Staubli VAL3: loadPage.pgx

program loadPage(string x_sPage, string& x_sItems[])
// load the next page
  local num i
begin
  // look if the page libload is correct
  i=page:libLoad(x_sPage)
  delay(0)
  logMsg("[VALPLAST] INTERFACE:PAGE LIBLOAD "+x_sPage+" result "+toString("",i))
  if i!=0
    popUpMsg("Loading page "+x_sPage+" error CODE "+toString("",i))
  else
    // copy all the field from x_sItems to the next page
    call use:stringCopy(x_sItems,page:sItems)
    call page:main()
    // to give back
    call use:stringCopy(page:sItems,x_sItems)
  endIf
end
